KUKA KRL data list: kuka_eki_hw_interface.dat

&ACCESS RVP
defdat kuka_eki_hw_interface
   ext bas(bas_command  :in,real  :in )
enddat
